(* PLC project PLC_DEV.project, CODESYS CODESYS V3.5 SP21 Patch 4 *)
(* stored: creationDateTime 2026-01-05T08:56:53.0725352, modificationDateTime 2026-01-05T08:56:50.7915579 *)

PROGRAM PLC_PRG
  VAR
    Counter : INT := 0;
    Toggle : BOOL := FALSE;
    BlinkTimer : TON;
    test : BOOL;
  END_VAR

                  
(* Increment counter every cycle *)
Counter := Counter + 1;

(* Toggle every 1 second *)
BlinkTimer(IN := TRUE, PT := T#1s);

IF BlinkTimer.Q THEN
    Toggle := NOT Toggle;
    BlinkTimer(IN := FALSE);
	test := FALSE;
END_IF
                
END_PROGRAM

CONFIGURATION Application
  RESOURCE Application ON PLC
    TASK MainTask(INTERVAL := T#20ms, PRIORITY := 1);
    PROGRAM PLC_PRG WITH MainTask : PLC_PRG;
  END_RESOURCE
END_CONFIGURATION
